FUNCTION GetZSide : LREAL
VAR_INPUT
	zPos : LREAL;
END_VAR
VAR
	zSide : LREAL;
	halfAreaWidth : LREAL;
END_VAR

halfAreaWidth := GVL_RobotArmConstants.PICKUP_AREA_WIDTH / 2;

IF (zPos < halfAreaWidth) THEN
	//Point is on the left side of the robot
	zSide := halfAreaWidth - zPos;
ELSE
	//Point is on the right side of the robot
	zSide := zPos - halfAreaWidth;
END_IF

GetZSide := zSide;

END_FUNCTION

(* stored: Version 1.1.0.1, ProductVersion 3.1.4024.12
   POU GetZSide: Id {3a2ca123-31f1-4d85-a5da-ba5f4030c5c1}, SpecialFunc None *)
